PROGRAM MAIN
VAR
	i : int;
END_VAR

i := i + 1;

END_PROGRAM

(* stored: Version 1.1.0.1, ProductVersion 3.1.4024.16
   POU MAIN: Id {708160a4-93d9-4013-9713-4347d7805f45}, SpecialFunc None *)
